{attribute 'GeneratedUsingTerminal: EL3001-0000-0017'}
{attribute addProperty BoxType "EL3001-0000-0017"}
{attribute addProperty Id "AI_StandardAT %I*AI_Standard_4A3944819WcStateAT %I*WcState_9091E0EB2InfoDataAT %I*InfoData_94A18F5E2"}
{attribute addProperty CRC "2975591319"}
{attribute addProperty Size "13"}
TYPE EL3001_B15BEB97 EXTENDS EtcSlaveTerminalBase_947E5A46 :
STRUCT
	{attribute addProperty Name "AI_Standard"}
	AI_Standard : AI_Standard_4A394481;
	{attribute addProperty Name "WcState"}
	WcState : WcState_9091E0EB;
	{attribute addProperty Name "InfoData"}
	InfoData : InfoData_94A18F5E;
END_STRUCT
END_TYPE

(* stored: Version 1.2.0.0, ProductVersion 3.1.4024.9
   DUT EL3001_B15BEB97: Id {c5450570-c7ce-42f2-a1f3-abb10245bec2} *)
